(* Logix 5000 project; controller CICD_test 1756-L85E rev 36.11; software revision 36.00 *)

TASK MainTask (continuous, watchdog 500 ms) : MainProgram

MODULES
   Local : 1756-L85E (ICP 0, rev 36.11)
END_MODULES

ADD_ON_INSTRUCTION AOI_Comparison   (* revision 1.0, ExecutePrescan *)
VAR_INPUT
   I_Parameter1 : DINT; {required}
   I_Parameter2 : DINT; {required}
END_VAR
VAR_OUTPUT
   O_Param1_grtr_than_Param2 : BOOL; {visible}
END_VAR

ROUTINE Logic   (* ladder *)
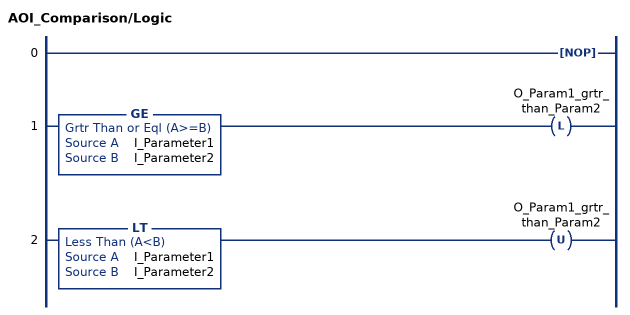
   0: NOP();
   1: GE(I_Parameter1,I_Parameter2)OTL(O_Param1_grtr_than_Param2);
   2: LT(I_Parameter1,I_Parameter2)OTU(O_Param1_grtr_than_Param2);
END_ROUTINE

ROUTINE Prescan   (* ladder *)
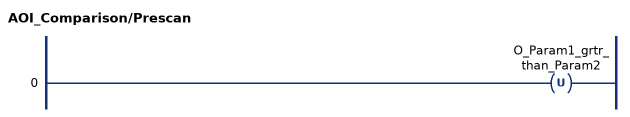
   0: OTU(O_Param1_grtr_than_Param2);
END_ROUTINE
END_ADD_ON_INSTRUCTION

ADD_ON_INSTRUCTION AOI_ModuleReset   (* revision 1.0 JDR *)
// Inhibits Module, Reset Module, Uninhibits Module
// Revision note:
// Developed for Safety I/O module reset with Signature/Lock
// Help:
// Inhibits Module, Reset Module, Uninhibits Module
// msg_Module_Reset can be shared by many modules, but must have Service Type = Device Reset
// The MSG path is set from IO_ModRef inside the AOI.
VAR_IN_OUT
   MSG_Module_Reset : MESSAGE; {required}   // Message Reset Module
   IO_ModRef : MODULE; {required}   // Module Reference
END_VAR
VAR_INPUT
   Cmd_Reset : BOOL; {required}   // Input Command To Run Routine
END_VAR
VAR_OUTPUT
   MSG_Err : BOOL; {access Read Only, visible}   // Message Error
   Mod_Flt : BOOL; {access Read Only, visible}   // Module Faulted
   Mod_Con : BOOL; {access Read Only, visible}   // Module Connecting
   Mod_Run : BOOL; {access Read Only, visible}   // Module Running
END_VAR
VAR
   ModulePath : SINT[82]; {access None}   // Module Path
   ONS : DINT; {access None}   // One Shot Array
   CardInhibit : DINT; {access None}   // Inhibit Value
   CardUnInhibit : DINT; {access None}   // UnInhibit Value
   Module_EntryStatus : DINT; {access None}   // Module Entry Status h1000 = Faulted h3000 = Connecting h4000 = Running h6000 = Inhibitted
   Reset_Run : BOOL; {access None}   // Run Reset Logic
   ModRun_TMR : TIMER := (PRE := 2000); {access None}   // Module Running Timer
   Mod_Inhibitted : BOOL; {access None}   // Module Inhibitted
END_VAR

ROUTINE Logic   (* ladder *)
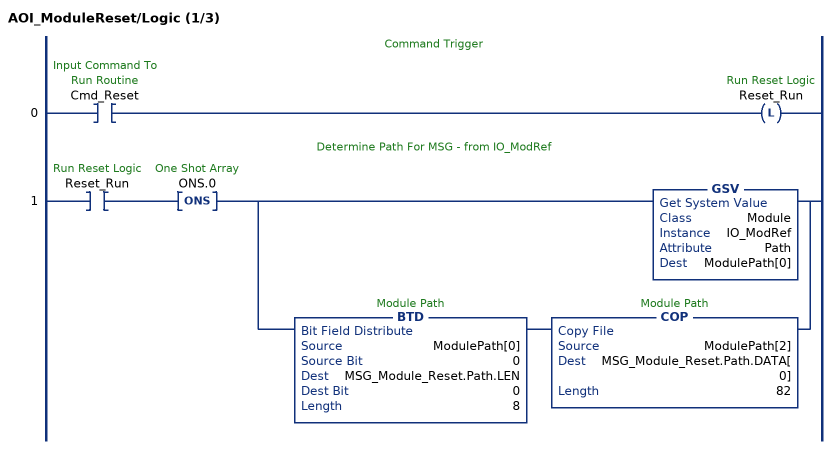
   // Command Trigger
   0: XIC(Cmd_Reset)OTL(Reset_Run);
   // Determine Path For MSG - from IO_ModRef
   1: XIC(Reset_Run)ONS(ONS.0)[GSV(Module,IO_ModRef,Path,ModulePath[0]) ,BTD(ModulePath[0],0,MSG_Module_Reset.Path.LEN,0,8) COP(ModulePath[2],MSG_Module_Reset.Path.DATA[0],82) ];
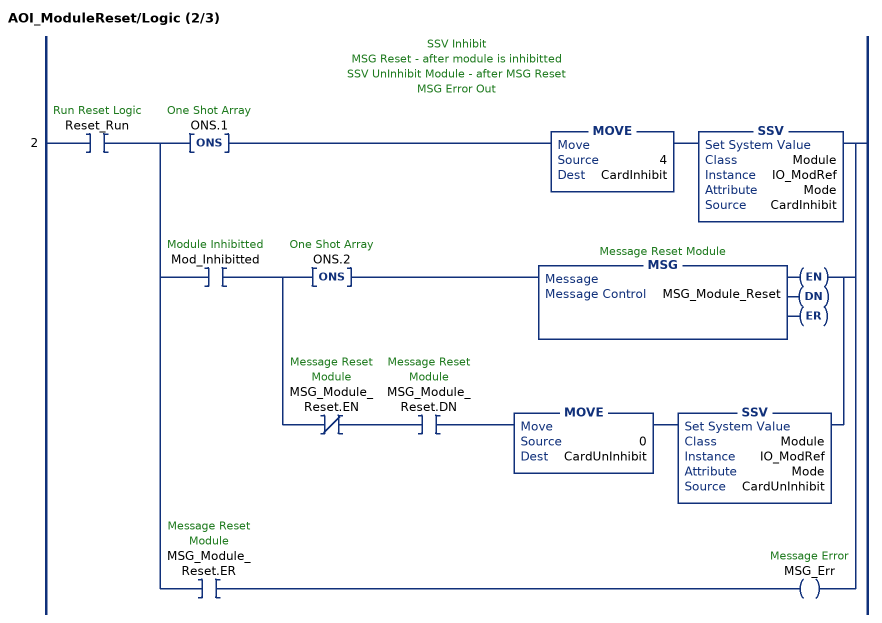
   // SSV Inhibit
   // MSG Reset - after module is inhibitted
   // SSV UnInhibit Module - after MSG Reset
   // MSG Error Out
   2: XIC(Reset_Run)[ONS(ONS.1) MOVE(4,CardInhibit) SSV(Module,IO_ModRef,Mode,CardInhibit) ,XIC(Mod_Inhibitted) [ONS(ONS.2) MSG(MSG_Module_Reset) ,XIO(MSG_Module_Reset.EN) XIC(MSG_Module_Reset.DN) MOVE(0,CardUnInhibit) SSV(Module,IO_ModRef,Mode,CardUnInhibit) ] ,XIC(MSG_Module_Reset.ER) OTE(MSG_Err) ];
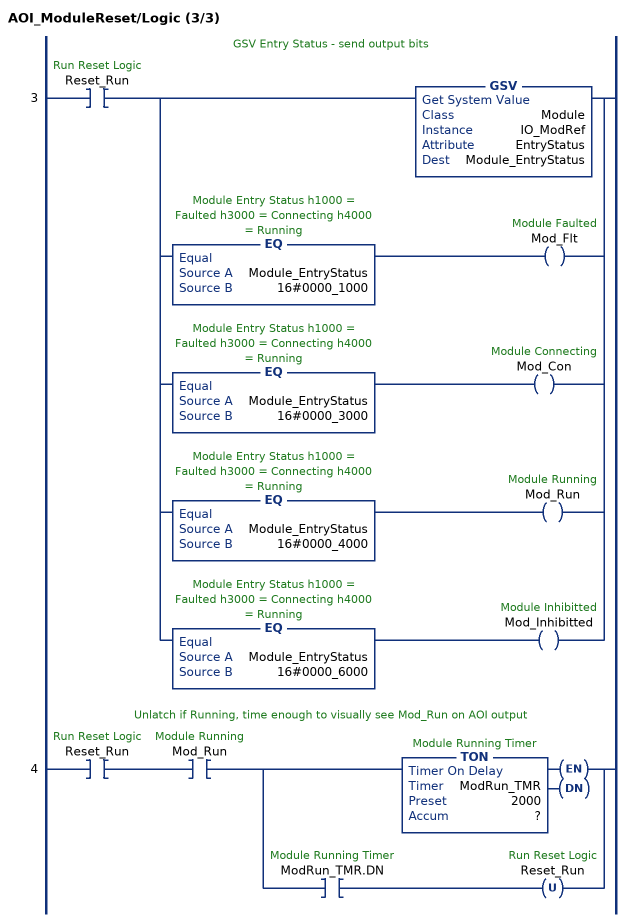
   // GSV Entry Status - send output bits
   3: XIC(Reset_Run)[GSV(Module,IO_ModRef,EntryStatus,Module_EntryStatus) ,EQ(Module_EntryStatus,16#0000_1000) OTE(Mod_Flt) ,EQ(Module_EntryStatus,16#0000_3000) OTE(Mod_Con) ,EQ(Module_EntryStatus,16#0000_4000) OTE(Mod_Run) ,EQ(Module_EntryStatus,16#0000_6000) OTE(Mod_Inhibitted) ];
   // Unlatch if Running, time enough to visually see Mod_Run on AOI output
   4: XIC(Reset_Run)XIC(Mod_Run)[TON(ModRun_TMR,?,?) ,XIC(ModRun_TMR.DN) OTU(Reset_Run) ];
END_ROUTINE
END_ADD_ON_INSTRUCTION

ADD_ON_INSTRUCTION WetBulbTemperature   (* revision 1.0, vendor Cardoso&Filho, ExecutePrescan *)
// This AOI calculates the Wet Bulb Temperature by using the Stull formula.
// Help:
// This AOI calculates the Wet Bulb Temperature by using the Stull formula.
// To minimise the processing required by the PLC, it uses look up tables for the Relative Humidity values.
VAR_INPUT
   Temperature : REAL; {required}   // Temperature input (if Fahrenheit used, please set correct tag)
   RelativeHumidity : REAL; {required}   // Relative Humidity input %
   isFahrenheit : BOOL; {required}   // 1 = Fahrenheit 0 = Celsius
END_VAR
VAR_OUTPUT
   WetBulbTemperature : REAL; {access Read Only, visible}   // Wet Bulb Temperature
END_VAR
VAR
   SecondTerm : REAL[101]; {access None}
   FirstTerm : REAL[101]; {access None}
   CelsiusTemperature : REAL; {access None}
   IntermediateCalc : REAL; {access None}
   DINT_RH : DINT; {access None}
   CelsiusWBTemperature : REAL; {access None}
END_VAR

ROUTINE Logic   (* structured text *)
   (*
   This AOI calculates the Wet Bulb Temperature by using the Stull formula.
   
   This was taken from the following website:
   
   https://www.omnicalculator.com/physics/wet-bulb
   
   To minimise the processing required by the PLC to do this calculation, the AOI resorts to using look up tables (that's why this takes so much memory).
   
   *)
   
   if isFahrenheit then
   	CelsiusTemperature := (Temperature-32.0)/1.8;
   else
   	CelsiusTemperature := Temperature;
   end_IF;
   DINT_RH := RelativeHumidity;
   
   // formula
   //  Tw = T * arctan[0.151977 * (rh% + 8.313659)^(1/2)] + arctan(T + rh%) - arctan(rh% - 1.676331) + 0.00391838 *(rh%)^(3/2) * arctan(0.023101 * rh%) - 4.686035
   //  This has been simplified to:
   //  Tw = T * FirstTerm[RH] + Intermediate Calc + SecondTerm[RH]
   //calculate the middle bit in the formula
   IntermediateCalc := ATAN(Temperature + RelativeHumidity);
   
   //calculate WetBulb Temperature
   CelsiusWBTemperature:= CelsiusTemperature * FirstTerm[DINT_RH] + IntermediateCalc + SecondTerm[DINT_RH];
   
   //update the output for the Imperial crowd
   if isFahrenheit then
   	WetBulbTemperature := (CelsiusWBTemperature*1.8)+32.0;
   else
   	WetBulbTemperature:=CelsiusWBTemperature;
   end_if;
   
END_ROUTINE

ROUTINE Prescan   (* structured text *)
// to put in place the correct parameters
   FirstTerm[0] := 0.412999183919456;
   FirstTerm[1] := 0.434276967500252;
   FirstTerm[2] := 0.454060080743169;
   FirstTerm[3] := 0.472556739086409;
   FirstTerm[4] := 0.489931226117599;
   FirstTerm[5] := 0.506315983562747;
   FirstTerm[6] := 0.521819708983603;
   FirstTerm[7] := 0.536532967729344;
   FirstTerm[8] := 0.550532195643151;
   FirstTerm[9] := 0.563882624999991;
   FirstTerm[10] := 0.576640469263689;
   FirstTerm[11] := 0.588854584963017;
   FirstTerm[12] := 0.60056775665652;
   FirstTerm[13] := 0.61181770498283;
   FirstTerm[14] := 0.622637887784856;
   FirstTerm[15] := 0.633058144240025;
   FirstTerm[16] := 0.643105218237873;
   FirstTerm[17] := 0.652803187721008;
   FirstTerm[18] := 0.662173819963356;
   FirstTerm[19] := 0.671236867912222;
   FirstTerm[20] := 0.680010319185341;
   FirstTerm[21] := 0.68851060670163;
   FirstTerm[22] := 0.696752787970507;
   FirstTerm[23] := 0.704750698586883;
   FirstTerm[24] := 0.712517084349741;
   FirstTerm[25] := 0.720063715551046;
   FirstTerm[26] := 0.727401486303549;
   FirstTerm[27] := 0.734540501243751;
   FirstTerm[28] := 0.741490151525149;
   FirstTerm[29] := 0.748259181681319;
   FirstTerm[30] := 0.754855748669075;
   FirstTerm[31] := 0.761287474184474;
   FirstTerm[32] := 0.767561491167731;
   FirstTerm[33] := 0.773684485268638;
   FirstTerm[34] := 0.779662731925439;
   FirstTerm[35] := 0.785502129612054;
   FirstTerm[36] := 0.791208229727168;
   FirstTerm[37] := 0.796786263530865;
   FirstTerm[38] := 0.802241166477608;
   FirstTerm[39] := 0.807577600246565;
   FirstTerm[40] := 0.812799972729915;
   FirstTerm[41] := 0.81791245620548;
   FirstTerm[42] := 0.82291900389095;
   FirstTerm[43] := 0.827823365052035;
   FirstTerm[44] := 0.832629098815608;
   FirstTerm[45] := 0.837339586820532;
   FirstTerm[46] := 0.841958044823116;
   FirstTerm[47] := 0.846487533360433;
   FirstTerm[48] := 0.850930967562922;
   FirstTerm[49] := 0.855291126197371;
   FirstTerm[50] := 0.859570660012408;
   FirstTerm[51] := 0.863772099450765;
   FirstTerm[52] := 0.867897861785706;
   FirstTerm[53] := 0.871950257732961;
   FirstTerm[54] := 0.875931497584199;
   FirstTerm[55] := 0.879843696903371;
   FirstTerm[56] := 0.88368888182311;
   FirstTerm[57] := 0.8874689939747;
   FirstTerm[58] := 0.891185895081857;
   FirstTerm[59] := 0.894841371245686;
   FirstTerm[60] := 0.898437136945561;
   FirstTerm[61] := 0.901974838778404;
   FirstTerm[62] := 0.90545605895674;
   FirstTerm[63] := 0.908882318584101;
   FirstTerm[64] := 0.912255080724649;
   FirstTerm[65] := 0.915575753282446;
   FirstTerm[66] := 0.918845691704414;
   FirstTerm[67] := 0.922066201519867;
   FirstTerm[68] := 0.925238540728373;
   FirstTerm[69] := 0.928363922046733;
   FirstTerm[70] := 0.931443515024981;
   FirstTerm[71] := 0.934478448040493;
   FirstTerm[72] := 0.937469810178549;
   FirstTerm[73] := 0.94041865300707;
   FirstTerm[74] := 0.943325992252588;
   FirstTerm[75] := 0.946192809384008;
   FirstTerm[76] := 0.949020053110182;
   FirstTerm[77] := 0.951808640796891;
   FirstTerm[78] := 0.954559459808375;
   FirstTerm[79] := 0.957273368778195;
   FirstTerm[80] := 0.959951198813862;
   FirstTerm[81] := 0.962593754639317;
   FirstTerm[82] := 0.96520181567909;
   FirstTerm[83] := 0.967776137087668;
   FirstTerm[84] := 0.970317450727362;
   FirstTerm[85] := 0.972826466097736;
   FirstTerm[86] := 0.975303871219448;
   FirstTerm[87] := 0.977750333475156;
   FirstTerm[88] := 0.980166500409975;
   FirstTerm[89] := 0.982553000493781;
   FirstTerm[90] := 0.984910443847533;
   FirstTerm[91] := 0.987239422935622;
   FirstTerm[92] := 0.989540513226143;
   FirstTerm[93] := 0.991814273820837;
   FirstTerm[94] := 0.994061248056375;
   FirstTerm[95] := 0.996281964078519;
   FirstTerm[96] := 0.998476935390616;
   FirstTerm[97] := 1.00064666137778;
   FirstTerm[98] := 1.00279162780807;
   FirstTerm[99] := 1.00491230731178;
   FirstTerm[100] := 1.0070091598401;
   
   SecondTerm[0] := -3.6531108341574;
   SecondTerm[1] := -4.09128101130617;
   SecondTerm[2] := -4.99855089843746;
   SecondTerm[3] := -5.60842606644933;
   SecondTerm[4] := -5.84754624814133;
   SecondTerm[5] := -5.95953661871908;
   SecondTerm[6] := -6.02161126211956;
   SecondTerm[7] := -6.05952030767856;
   SecondTerm[8] := -6.08379123547508;
   SecondTerm[9] := -6.09943992136132;
   SecondTerm[10] := -6.10913407129205;
   SecondTerm[11] := -6.11441266150827;
   SecondTerm[12] := -6.11622046037205;
   SecondTerm[13] := -6.11516667697321;
   SecondTerm[14] := -6.11166024379888;
   SecondTerm[15] := -6.10598513983822;
   SecondTerm[16] := -6.09834452933237;
   SecondTerm[17] := -6.08888774639591;
   SecondTerm[18] := -6.07772738789046;
   SecondTerm[19] := -6.06495046880874;
   SecondTerm[20] := -6.05062588863923;
   SecondTerm[21] := -6.03480953623053;
   SecondTerm[22] := -6.01754784316729;
   SecondTerm[23] := -5.99888029447187;
   SecondTerm[24] := -5.97884122460011;
   SecondTerm[25] := -5.95746111505514;
   SecondTerm[26] := -5.93476753927376;
   SecondTerm[27] := -5.91078585468354;
   SecondTerm[28] := -5.88553971158705;
   SecondTerm[29] := -5.85905142816312;
   SecondTerm[30] := -5.83134226692107;
   SecondTerm[31] := -5.80243263823249;
   SecondTerm[32] := -5.7723422497084;
   SecondTerm[33] := -5.74109021528467;
   SecondTerm[34] := -5.70869513432806;
   SecondTerm[35] := -5.6751751484777;
   SecondTerm[36] := -5.64054798201802;
   SecondTerm[37] := -5.60483097015052;
   SecondTerm[38] := -5.56804107845941;
   SecondTerm[39] := -5.53019491605745;
   SecondTerm[40] := -5.49130874428476;
   SecondTerm[41] := -5.45139848236587;
   SecondTerm[42] := -5.41047971107395;
   SecondTerm[43] := -5.36856767517859;
   SecondTerm[44] := -5.32567728524447;
   SecondTerm[45] := -5.28182311918963;
   SecondTerm[46] := -5.23701942389009;
   SecondTerm[47] := -5.19128011702566;
   SecondTerm[48] := -5.14461878929223;
   SecondTerm[49] := -5.09704870705358;
   SecondTerm[50] := -5.04858281546752;
   SecondTerm[51] := -4.99923374209295;
   SecondTerm[52] := -4.94901380096437;
   SecondTerm[53] := -4.89793499710682;
   SecondTerm[54] := -4.84600903145481;
   SecondTerm[55] := -4.79324730613358;
   SecondTerm[56] := -4.739660930058;
   SecondTerm[57] := -4.6852607248036;
   SecondTerm[58] := -4.63005723070492;
   SecondTerm[59] := -4.5740607131378;
   SecondTerm[60] := -4.51728116894469;
   SecondTerm[61] := -4.45972833296467;
   SecondTerm[62] := -4.40141168463302;
   SecondTerm[63] := -4.34234045461819;
   SecondTerm[64] := -4.28252363146719;
   SecondTerm[65] := -4.22196996823365;
   SecondTerm[66] := -4.16068798906535;
   SecondTerm[67] := -4.09868599573142;
   SecondTerm[68] := -4.03597207407149;
   SecondTerm[69] := -3.9725541003518;
   SecondTerm[70] := -3.90843974751561;
   SecondTerm[71] := -3.84363649131689;
   SecondTerm[72] := -3.77815161632872;
   SecondTerm[73] := -3.71199222181899;
   SecondTerm[74] := -3.64516522748777;
   SecondTerm[75] := -3.57767737906207;
   SecondTerm[76] := -3.50953525374477;
   SecondTerm[77] := -3.44074526551568;
   SecondTerm[78] := -3.37131367028359;
   SecondTerm[79] := -3.30124657088888;
   SecondTerm[80] := -3.2305499219571;
   SecondTerm[81] := -3.15922953460459;
   SecondTerm[82] := -3.08729108099734;
   SecondTerm[83] := -3.01474009876535;
   SecondTerm[84] := -2.94158199527454;
   SecondTerm[85] := -2.8678220517589;
   SecondTerm[86] := -2.7934654273158;
   SecondTerm[87] := -2.71851716276739;
   SecondTerm[88] := -2.64298218439145;
   SecondTerm[89] := -2.5668653075249;
   SecondTerm[90] := -2.49017124004356;
   SecondTerm[91] := -2.41290458572153;
   SecondTerm[92] := -2.33506984747377;
   SecondTerm[93] := -2.25667143048545;
   SecondTerm[94] := -2.17771364523156;
   SecondTerm[95] := -2.09820071039039;
   SecondTerm[96] := -2.01813675565421;
   SecondTerm[97] := -1.93752582444074;
   SecondTerm[98] := -1.85637187650874;
   SecondTerm[99] := -1.77467879048101;
   SecondTerm[100] := -1.69245036627809;
   
END_ROUTINE
END_ADD_ON_INSTRUCTION

VAR_GLOBAL   (* controller tags *)
   AOI_WetBulbTemp : WetBulbTemperature;
   test_BOOL : BOOL;
   test_DINT_1 : DINT := 2;
   test_DINT_2 : DINT := 20;
   test_DINT_3 : DINT := 30;
   test_STRING : STRING;
END_VAR

PROGRAM MainProgram   (* main routine MainRoutine *)

ROUTINE MainRoutine   (* ladder *)
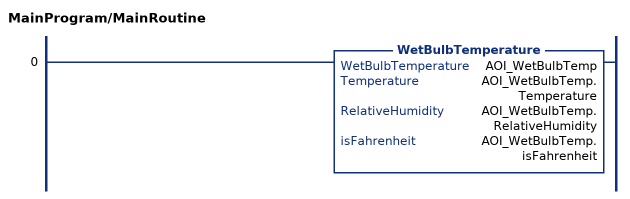
   0: WetBulbTemperature(AOI_WetBulbTemp,AOI_WetBulbTemp.Temperature,AOI_WetBulbTemp.RelativeHumidity,AOI_WetBulbTemp.isFahrenheit);
END_ROUTINE
END_PROGRAM
